FUNCTION_BLOCK FB_ExecutorTreeSearch
VAR_INPUT
END_VAR
VAR_OUTPUT
END_VAR
VAR
	_observer : InterfaceObserver;
END_VAR

METHOD search : BOOL
VAR_INPUT
	executor : REFERENCE TO FB_Executor;
END_VAR
VAR
	_child_executor  : REFERENCE TO FB_Executor;
	_all_done : BOOL;
END_VAR
_all_done := TRUE;
IF NOT _observer.subscribe_job_directory(executor) THEN
	_all_done := FALSE;
END_IF

// Recursive process if child object exists.
IF executor.children <> 0 THEN
	REPEAT 
		_child_executor REF= executor.children.each_executor;
		IF __ISVALIDREF(_child_executor) THEN
			IF NOT THIS^.search(_child_executor) THEN
				_all_done := FALSE;
			END_IF
		END_IF
	UNTIL
		NOT __ISVALIDREF(_child_executor)
	END_REPEAT	
END_IF
search := _all_done;
END_METHOD

PROPERTY subscriber : InterfaceObserver
SET
_observer := subscriber;
END_SET
END_PROPERTY

END_FUNCTION_BLOCK

(* stored: Version 1.1.0.1, ProductVersion 3.1.4024.12
   POU FB_ExecutorTreeSearch: Id {149b5315-e5ca-4a5c-b083-4e295a6fbba5}, SpecialFunc None
   Method search: Id {4aa60b52-b4c1-49ad-bcc1-ddd28e76b7fb}
   Property subscriber: Id {cbd9a383-4bd6-4f9d-9073-4f772a89385d}
   Set Set: Id {bc01bd66-0598-4f1e-9c20-0e70382077be} *)
